PROGRAM B_4_3_PRG_Master_SlideNest

VAR


/////////////////////////////////////////////////////////////////////////////////////I O/////////////////////////////////////////////////////////////////////////////////////	
	
	bNestRight							: BOOL;
	bNestLeft							: BOOL;
	bNestRightHMI						: BOOL;
	bLeftRightHMI						: BOOL;
	bNestInLeftPos						: BOOL;
	bNestInRightPos						: BOOL;
	
	bProcessCylinderUp					: BOOL;
	bProcessDoorClosed					: BOOL;

	

	
	
END_VAR

d_ACT_Set_Events_Station_4B();
a_ACT_Ctrl_Station_4B();
b_ACT_IO_B();

ACTION a_ACT_Ctrl_Station_4B:
/////////////////////////////////////////////////////////////////////////////////////UTILITIES/////////////////////////////////////////////////////////////////////////////////////

/////////////////////////////////////////////////////////////////////////////////////CONDITIONS/////////////////////////////////////////////////////////////////////////////////////


IF stSlideNest.CMD.bAbort THEN
	
	stSlideNest.State												:= E_SlideNest_State.RESET;
	
ELSIF stSlideNest.CMD.bEndCycle THEN
	
	stSlideNest.State												:= E_SlideNest_State.STOPPING;

END_IF

CASE stSlideNest.State OF
	
	E_SlideNest_State.ABORTED:
	
								IF stSlideNest.CMD.bEnable  THEN
									
									stSlideNest.State				:= E_SlideNest_State.HOMING;
								
								END_IF
								
	E_SlideNest_State.HOMING: 
								
								IF bProcessDoorClosed AND bProcessCylinderUp THEN
									
									bNestLeft							:= TRUE;
									
								END_IF
								
								
								IF bNestInLeftPos THEN
									
									stSlideNest.State				:= E_SlideNest_State.READY;									
									bNestLeft						:= FALSE;
																	
								END_IF
	
	
	E_SlideNest_State.READY:
	
								IF stSlideNest.CMD.bExecute AND 	stSlideNest.CMD.SlideCylinderCMD.MoveRight	THEN

									stSlideNest.State				:= E_SlideNest_State.MOVE_RIGHT;
									
								ELSIF stSlideNest.CMD.bExecute AND 	stSlideNest.CMD.SlideCylinderCMD.MoveLeft	THEN
									
									stSlideNest.State				:= E_SlideNest_State.MOVE_LEFT;									
																		
								END_IF
	

	E_SlideNest_State.MOVE_RIGHT:
	
								bNestRight							:= TRUE;
								
								IF bNestInRightPos	THEN
									
									stSlideNest.State				:= E_SlideNest_State.DONE;
								
								END_IF
								
	E_SlideNest_State.MOVE_LEFT:
	
								bNestLeft							:= TRUE;
								
								IF bNestInLeftPos THEN
									
									stSlideNest.State				:= E_SlideNest_State.DONE;
								
								END_IF
								
	E_SlideNest_State.DONE:
	
	
								IF stSlideNest.CMD.bAcknowledge THEN
									
									stSlideNest.CMD.bAcknowledge	:= FALSE;
									stSlideNest.State				:= E_SlideNest_State.RESET;
								
								END_IF
	
	
	E_SlideNest_State.RESET:	
	
								bNestRight							:= FALSE;
								bNestLeft							:= FALSE;
								
								IF NOT stSlideNest.CMD.bAbort AND NOT stSlideNest.CMD.bEndCycle THEN
									
									stSlideNest.State				:= E_SlideNest_State.READY;
									
								ELSE stSlideNest.State			:= E_SlideNest_State.ABORTED;
								END_IF
									

ELSE stSlideNest.State		:= E_SlideNest_State.ABORTED;
	
END_CASE
/////////////////////////////////////////////////////////////////////////////////////STATUS/////////////////////////////////////////////////////////////////////////////////////

stSlideNest.Status.bBusy			:= 	stSlideNest.State	= E_SlideNest_State.MOVE_RIGHT OR
										stSlideNest.State	= E_SlideNest_State.MOVE_LEFT OR 
										stSlideNest.State	= E_SlideNest_State.STOPPING OR
										stSlideNest.State	= E_SlideNest_State.HOMING;
								
stSlideNest.Status.bDone			:=	stSlideNest.State	= E_SlideNest_State.DONE;

stSlideNest.Status.bReady			:= 	stSlideNest.State	= E_SlideNest_State.READY;

stSlideNest.Status.bStopped		:= 	NOT stSlideNest.Status.bBusy;
END_ACTION

ACTION b_ACT_IO_B:

bNestInLeftPos									:= dw_T08_EL1809.iSlideNestRetracted;
bNestInRightPos									:= dw_T08_EL1809.iSlideNestExtended; 

IF bNestRight OR bSlideNestRight AND bProcessCylinderUp THEN
	
	dw_T09_EL2809.qExtendSlideNest	:= TRUE ;
	dw_T09_EL2809.qRetractSlideNest	:= FALSE;

ELSIF bNestLeft OR bSlideNestLeft AND bProcessCylinderUp THEN
	
	dw_T09_EL2809.qExtendSlideNest	:= FALSE;
	dw_T09_EL2809.qRetractSlideNest	:= TRUE;
	
ELSIF stMachineStatus.bFault THEN
	
	dw_T09_EL2809.qExtendSlideNest	:= FALSE;
	dw_T09_EL2809.qRetractSlideNest	:= FALSE;

END_IF

bProcessCylinderUp								:= stTwinSAFE.qProcessCylinderRetracted;

bProcessDoorClosed 								:= dw_T05_EL1918.iProcessDoorClosed1 AND dw_T05_EL1918.iProcessDoorClosed2 AND dw_T05_EL1918.iProcessDoorFB;
END_ACTION

ACTION d_ACT_Set_Events_Station_4B:
//IMMEDIATE FAULTS

stStationEvents[5].aEvents[0].bEventTimer( IN :=  (bNestLeft OR bSlideNestLeft) AND NOT bNestInLeftPos, PT := T#3S);
stStationEvents[5].aEvents[0].bFault						:= TRUE;
stStationEvents[5].aEvents[0].bEventFlag					:= stStationEvents[5].aEvents[0].bEventTimer.Q;
stStationEvents[5].aEvents[0].bEventText					:= 'Slide Nest  Retract timeout';
stStationEvents[5].aEvents[0].sSolution						:= 'Check Nest Cylinder, neumatic connections and sensors';

stStationEvents[5].aEvents[1].bEventTimer( IN :=  (bNestRight  OR bSlideNestRight) AND NOT bNestInRightPos, PT := T#3S);
stStationEvents[5].aEvents[1].bFault						:= TRUE;
stStationEvents[5].aEvents[1].bEventFlag					:= stStationEvents[5].aEvents[1].bEventTimer.Q;
stStationEvents[5].aEvents[1].bEventText					:= 'Slide Nest Extend timeout';
stStationEvents[5].aEvents[1].sSolution						:= 'Check Nest Cylinder, neumatic connections and sensors ';
END_ACTION

END_PROGRAM

(* stored: Version 1.1.0.1, ProductVersion 3.1.4026.18
   POU B_4_3_PRG_Master_SlideNest: Id {23f0e1e1-7563-491f-bb2c-a8937b7ea92f}, SpecialFunc None
   Action a_ACT_Ctrl_Station_4B: Id {4fcc76fc-a9f9-4009-ab38-1acad5f7752c}
   Action b_ACT_IO_B: Id {7592d3e9-dd86-422c-8792-e5f14744b8ea}
   Action d_ACT_Set_Events_Station_4B: Id {938e0a0a-091d-495e-86ce-4b8a012a211a} *)
